FUNCTION_BLOCK E_TRIG (* Trigger unconnected input events of the specified type inside a resource *)
  (* Standard: 61499-2 *)
  (* Version 1.0, 2025-01-08, Mario Kastner *)
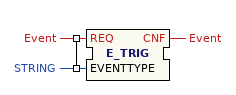
  EVENT_INPUT
    REQ WITH EVENTTYPE; (* Request trigger of unconnected event pins of type EVENTTYPE *)
  END_EVENT
  EVENT_OUTPUT
    CNF; (* Confirmation of Requested Service *)
  END_EVENT
  VAR_INPUT
    EVENTTYPE : STRING := 'EInit'; (* Event type to be triggered *)
  END_VAR
END_FUNCTION_BLOCK
